{attribute 'qualified_only'}
{attribute 'strict'}
TYPE ControlInterfaceType :
(
  Undefined,
  Position, // Position-control: Full control over the entire kinematic state (Default)
  Velocity // Velocity-control: Ignores the current position, target position, and velocity limits
);
END_TYPE

(* stored: Version 1.1.0.1
   DUT ControlInterfaceType: Id {fa41777e-c926-434f-898a-1e6e98888ce1} *)
